Staubli VAL3: dataGet.pgx

program dataGet()
begin
  //dataGet essentially gathers all of the inputs together and then calls the appropiate method
  //It is VITAL that the signal sent ends in either a ) (gesture) and } (movement).
  sBuffer = chr(nBuffer)
  putln(sBuffer)
  if(sBuffer == ")")
    //putln("dataGet")
    call actGesture()
    sInput = ""
    nBuffer = 0
    sBuffer = ""
  elseIf(sBuffer == "}")
    //putln(sInput)
    call parseMovement()
    //sInput = ""
  else
    sInput = sInput + sBuffer
  endIf
  //sBuffer = ""
end
